PROGRAM MAIN
VAR
	
END_VAR

GVL_General.fbAxis();


GVL_General.fbAxis.PowerOn();
GVL_General.bPowrOn :=  GVL_General.Axis1.NcToPlc.StateDWord.20;

GVL_General.fbAxis.Stop();

IF GVL_General.bPowrOn THEN 
	GVL_General.fbAxis.MoveVelocity();
	GVL_General.fbAxis.MoveRelative();	
END_IF

GVL_General.fbAxis.SetPosition();

GVL_General.hmiLActPos := GVL_General.Axis1.NcToPlc.ActPos;

GVL_General.fbAxis.SetPosition();

IF GVL_General.bPowrOn AND GVL_General.hmiManualJog THEN 
	GVL_General.fbAxis.Jog();	
END_IF

END_PROGRAM

(* stored: Version 1.1.0.1, ProductVersion 3.1.4022.16
   POU MAIN: Id {6b59d043-3d9d-40bc-ba8d-a42acc712532}, SpecialFunc None *)
